FUNCTION F_AnalogIn : REAL
VAR_INPUT
	Input																: INT;
	Low																	: REAL;
	High																: REAL;
	Minimum																: REAL;
	Offset																: REAL;
END_VAR
VAR
	Value																: REAL;
END_VAR

// F_AnalogIn
// Rev 1.0 - December 28, 2023

Value																	:= ((High - Low) / 32767.0) * INT_TO_REAL(Input) + Low;		// Determine output based on scale
Value																	:= Value + Offset;											// Adjust for any user offset
F_AnalogIn																:= SEL(ABS(Value) > Minimum, 0, Value);						// Value must be above (or below, if negative) minimum or zero is returned

END_FUNCTION

(* stored: Version 1.1.0.1, ProductVersion 3.1.4024.12
   POU F_AnalogIn: Id {983d5a87-6711-44c6-87e2-607ffb4f42dd}, SpecialFunc None *)
